FUNCTION_BLOCK PUBLIC FB_TrafficLight
VAR
	tRedDuration: TIME := T#6S;
	tYellowDuration: TIME := T#2S;
	tGreenDuration: TIME := T#4S;
	
	fbTon: TON;
	
	RedLight: BOOL;
	YellowLight: BOOL;
	GreenLight: BOOL;
	
	nStep: SINT := 0;
	bStart: BOOL := FALSE;
	bSwitach: BOOL := FALSE;
END_VAR

IF bStart THEN
	CASE nStep OF
		0: (* GREEN *)
			TurnOnLight(E_Light.Green);
			fbTon(IN := TRUE, PT := tGreenDuration);
			IF fbTon.Q THEN
				fbTon(IN := FALSE);
				nStep := 1;
			END_IF
		1: (* YELLOW *)
			TurnOnLight(E_Light.Yellow);
			fbTon(IN := TRUE, PT := tYellowDuration);
			IF fbTon.Q THEN
				fbTon(IN := FALSE);
				nStep := 2;
				bSwitach := TRUE;
			END_IF
		2: (* RED *)
			TurnOnLight(E_Light.Red);
			fbTon(IN := TRUE, PT := tRedDuration);
			IF fbTon.Q THEN
				fbTon(IN := FALSE);
				nStep := 0;
				bStart := FALSE;
			END_IF
	END_CASE
ELSE
	TurnOnLight(E_Light.Red);
END_IF

METHOD PUBLIC CanSwitch : BOOL
VAR
	bReturn: BOOL := FALSE;
END_VAR
IF bSwitach THEN
	bReturn := TRUE;
	bSwitach := FALSE;
END_IF
CanSwitch := bReturn;
END_METHOD

METHOD PUBLIC Setup
VAR_INPUT
	redDuration: TIME;
	yellowDuration: TIME;
	greenDuration: TIME;
END_VAR
tRedDuration := redDuration;
tYellowDuration := yellowDuration;
tGreenDuration := greenDuration;
END_METHOD

PROPERTY PUBLIC Start : BOOL
GET
Start := bStart;
END_GET
SET
bStart := Start;
END_SET
END_PROPERTY

METHOD PRIVATE TurnOnLight
VAR_INPUT
	eLight: E_Light;
END_VAR
CASE eLight OF
	E_Light.Red:
		IF NOT RedLight THEN
			RedLight := TRUE;
			YellowLight := FALSE;
			GreenLight := FALSE;
		END_IF 

	E_Light.Yellow:
		IF NOT YellowLight THEN
			RedLight := FALSE;
			YellowLight := TRUE;
			GreenLight := FALSE;
		END_IF 

	
	E_Light.Green:
		IF NOT GreenLight THEN
			RedLight := FALSE;
			YellowLight := FALSE;
			GreenLight := TRUE;
		END_IF 

	ELSE
		RedLight := FALSE;
		YellowLight := FALSE;
		GreenLight := FALSE;
END_CASE
END_METHOD

END_FUNCTION_BLOCK

(* stored: Version 1.1.0.1, ProductVersion 3.1.4024.12
   POU FB_TrafficLight: Id {81f779f5-7b76-4f95-b1bf-c39a496d423c}, SpecialFunc None
   Method CanSwitch: Id {e2f04201-4b0b-4fe6-b32c-2397e884ea61}
   Method Setup: Id {9d28cf18-c69a-4ced-b8e7-9ebfa135b382}
   Property Start: Id {5a072ebf-81f9-45f9-b2ea-6a55a74c44d6}
   Get Get: Id {6a7a06fd-c816-42d2-9f3e-b289aec12aef}
   Set Set: Id {23f109f4-38da-4ede-a4bf-fbfee4ec65db}
   Method TurnOnLight: Id {281268d3-fc86-4842-9db5-5565e552e7bd} *)
